// TIA Portal V19 export
DATA_BLOCK "HMIGraphicControl_DB"   // DB21
// stored: AutoNumber false, InstanceOfName HMIGraphicControl, InstanceOfType FB
"HMIGraphicControl"
   // VAR_INPUT
   //    "Conveyor Speed" { ExternalAccessible := 'False'; ExternalVisible := 'False'; ExternalWritable := 'False'} : Real;
   //    "Arm Speed" { ExternalAccessible := 'False'; ExternalVisible := 'False'; ExternalWritable := 'False'} : Real;
   //    "Conveyor Max Speed" { ExternalAccessible := 'False'; ExternalVisible := 'False'; ExternalWritable := 'False'} : Real;
   //    "Arm Max Speed" { ExternalAccessible := 'False'; ExternalVisible := 'False'; ExternalWritable := 'False'} : Real;
   //    ConveyorMoving : Bool;
   //    ArmMoving : Bool;
   //    Reset : Bool;
   // END_VAR
   // VAR_OUTPUT
   //    Conveyor_On : Bool;
   //    Arm_On : Bool;
   // END_VAR
   // VAR_IN_OUT
   //    System_Enable : Bool;
   //    Graphic_Index { ExternalAccessible := 'False'; ExternalVisible := 'False'; ExternalWritable := 'False'} : Int;
   //    Box_Cnt : DInt;
   //    Pallet_Cnt : DInt;
   // END_VAR
   // VAR
   //    IEC_Timer_0_Instance { S7_SetPoint := 'True'} : IEC_TIMER;
   //    ConveyorTick : Bool;
   //    ConveyorTime : DInt;
   //    ConveyorTimeFactor : DInt;
   //    ArmTick : Bool;
   //    ArmTimeFactor : DInt;
   //    ArmTime : DInt;
   //    IEC_Timer_0_Instance_1 { S7_SetPoint := 'True'} : IEC_TIMER;
   // END_VAR
BEGIN
END_DATA_BLOCK
